// Mitsubishi GX Works2 project: GX W2 CA DK C   PLC: FX3G

// global labels: Global1
VAR_GLOBAL
  iStart_PB AT X001 : BOOL;
  iStop_PB AT X002 : BOOL;
  oExtraction_Fan AT Y001 : BOOL;
  oFan_On_Lamp AT Y002 : BOOL;
  oFan_Service_Due AT Y003 : BOOL;
  iReset_PB AT X003 : BOOL;
END_VAR

// task Task_01 (event TRUE, interval 0, priority 31): POU_01

PROGRAM POU_01
VAR
  bSystem_Started : BOOL;
  TON_1 : TON;
  CTU_1 : CTU;
END_VAR
(* structured ladder/FBD written out as ST: instructions are called as NAME(EN, inputs, outputs); _pN, _eN, _tN stand for wires *)
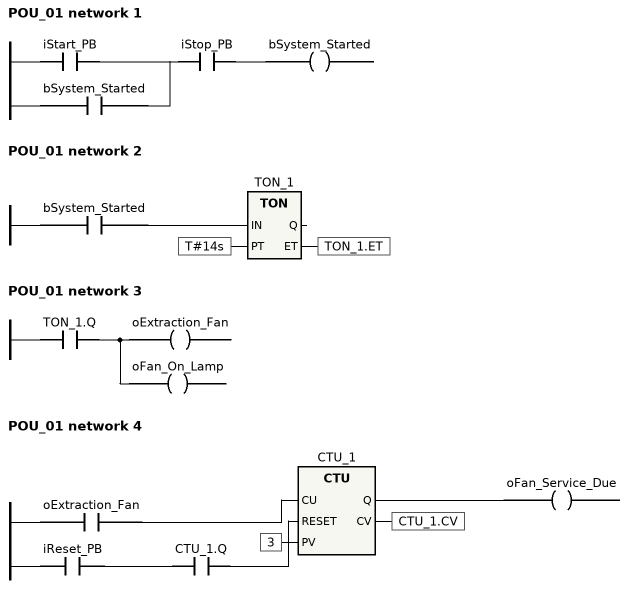
(* network 1 *)
bSystem_Started := (iStart_PB OR bSystem_Started) AND iStop_PB;
(* network 2 *)
TON_1(IN := bSystem_Started, PT := T#14s, ET => TON_1.ET);
(* network 3 *)
oExtraction_Fan := TON_1.Q;
oFan_On_Lamp := TON_1.Q;
(* network 4 *)
CTU_1(CU := oExtraction_Fan, RESET := iReset_PB AND CTU_1.Q, PV := 3, CV => CTU_1.CV);
oFan_Service_Due := CTU_1.Q;
END_PROGRAM
